// Mitsubishi GX Works2 project: ex2automation   PLC: FX3G

// global labels: Global1
VAR_GLOBAL
  start_switch AT X007 : BOOL;
  workday_start AT Y000 : BOOL;
  kill_switch AT X005 : BOOL;
  oatmeal_overr AT M0 : BOOL;
  protein_over AT M1 : BOOL;
  honey_over AT M2 : BOOL;
  dayover AT M3 : BOOL;
  daylight AT Y000 : BOOL;
  input_quantities AT X003 : BOOL;
  typeOfSnack AT X003 : BOOL;
END_VAR
VAR_GLOBAL CONSTANT
  const1 : INT := 2000;
END_VAR
VAR_GLOBAL
  normal_Snack AT M4 : BOOL;
  reset : BOOL;
  reset_Button AT M69 : BOOL;
  hold_Normal AT M41 : BOOL;
END_VAR
VAR_GLOBAL CONSTANT
  const2 : INT := 4000;
END_VAR
VAR_GLOBAL
  protein_Snack AT M5 : BOOL;
  hold_Protein AT M51 : BOOL;
  input_Oatmeal AT D1111 : REAL;
  oatmeal_Inv AT D1122 : REAL;
  input_protein AT D2222 : REAL;
  protein_Inv AT D2233 : REAL;
  input_Honey AT D3333 : REAL;
  honey_Inv AT D3344 : REAL;
  analog_input2 AT D8280 : INT;
END_VAR
VAR_GLOBAL CONSTANT
  const3 : REAL := 400;
  const4 : REAL := 320;
  const6 : REAL := 400;
  const7 : REAL := 320;
  const8 : REAL := 160;
  const9 : INT := 120;
END_VAR
VAR_GLOBAL
  start_shake_normal AT M10 : BOOL;
  start_shake_special AT M11 : BOOL;
  shakeTimer AT TC1 : BOOL;
END_VAR
VAR_GLOBAL CONSTANT
  shakeTimeValue : INT := 50;
END_VAR
VAR_GLOBAL
  timer_shake AT TS1 : BOOL;
  mixing_light AT Y003 : BOOL;
END_VAR
VAR_GLOBAL CONSTANT
  const5 : REAL := 160;
END_VAR
VAR_GLOBAL
  oatmeal_ok_n AT M42 : BOOL;
  protein_ok_n AT M43 : BOOL;
  honey_ok_n AT M44 : BOOL;
END_VAR
VAR_GLOBAL CONSTANT
  const0 : INT;
END_VAR
VAR_GLOBAL
  oatmeal_ok_p AT M52 : BOOL;
  protein_ok_p AT M53 : BOOL;
  honey_ok_p AT M54 : BOOL;
  func_reset AT M99 : BOOL;
  typeOfSnackHelp AT M33 : BOOL;
  hold_Shake AT M110 : BOOL;
  Bake_start AT X002 : BOOL;
  Bake_normal AT TC2 : BOOL;
  Bake_Protein AT TC3 : BOOL;
END_VAR
VAR_GLOBAL CONSTANT
  normalBakingTime : INT := 40;
  proteinBakingTime : INT := 50;
END_VAR
VAR_GLOBAL
  Baking_timer_normal AT TS2 : BOOL;
  Baking_timer_protein AT TS3 : BOOL;
  Bake_blink_help AT M60 : BOOL;
  blinkLight1 AT TC5 : BOOL;
END_VAR
VAR_GLOBAL CONSTANT
  blink_const : INT := 2;
END_VAR
VAR_GLOBAL
  blinktimer1 AT TS5 : BOOL;
  blinking_light1 AT Y001 : BOOL;
  blinkLight2 AT TC6 : BOOL;
  blinktime2 AT TS6 : BOOL;
  blinking_light2 AT Y002 : BOOL;
  packing_start AT X006 : BOOL;
  single_pack AT X000 : BOOL;
  light_help AT M61 : BOOL;
  packCounter AT CC1 : BOOL;
END_VAR
VAR_GLOBAL CONSTANT
  packconstant : INT := 8;
END_VAR
VAR_GLOBAL
  outPackCounter AT CS1 : BOOL;
  packinglight AT Y004 : BOOL;
END_VAR
VAR_GLOBAL CONSTANT
  const11 : INT := 1;
END_VAR
VAR_GLOBAL
  finishPackage AT D4444 : INT;
END_VAR
VAR_GLOBAL CONSTANT
  const12 : INT := 40;
END_VAR
VAR_GLOBAL
  analog_output AT D8282 : INT;
  reset_help AT M70 : BOOL;
  hold_bake_start AT M22 : BOOL;
END_VAR

// task Task_01 (event TRUE, interval 0, priority 31): POU_01

PROGRAM POU_01
(* structured ladder/FBD written out as ST: instructions are called as NAME(EN, inputs, outputs); _pN, _eN, _tN stand for wires *)
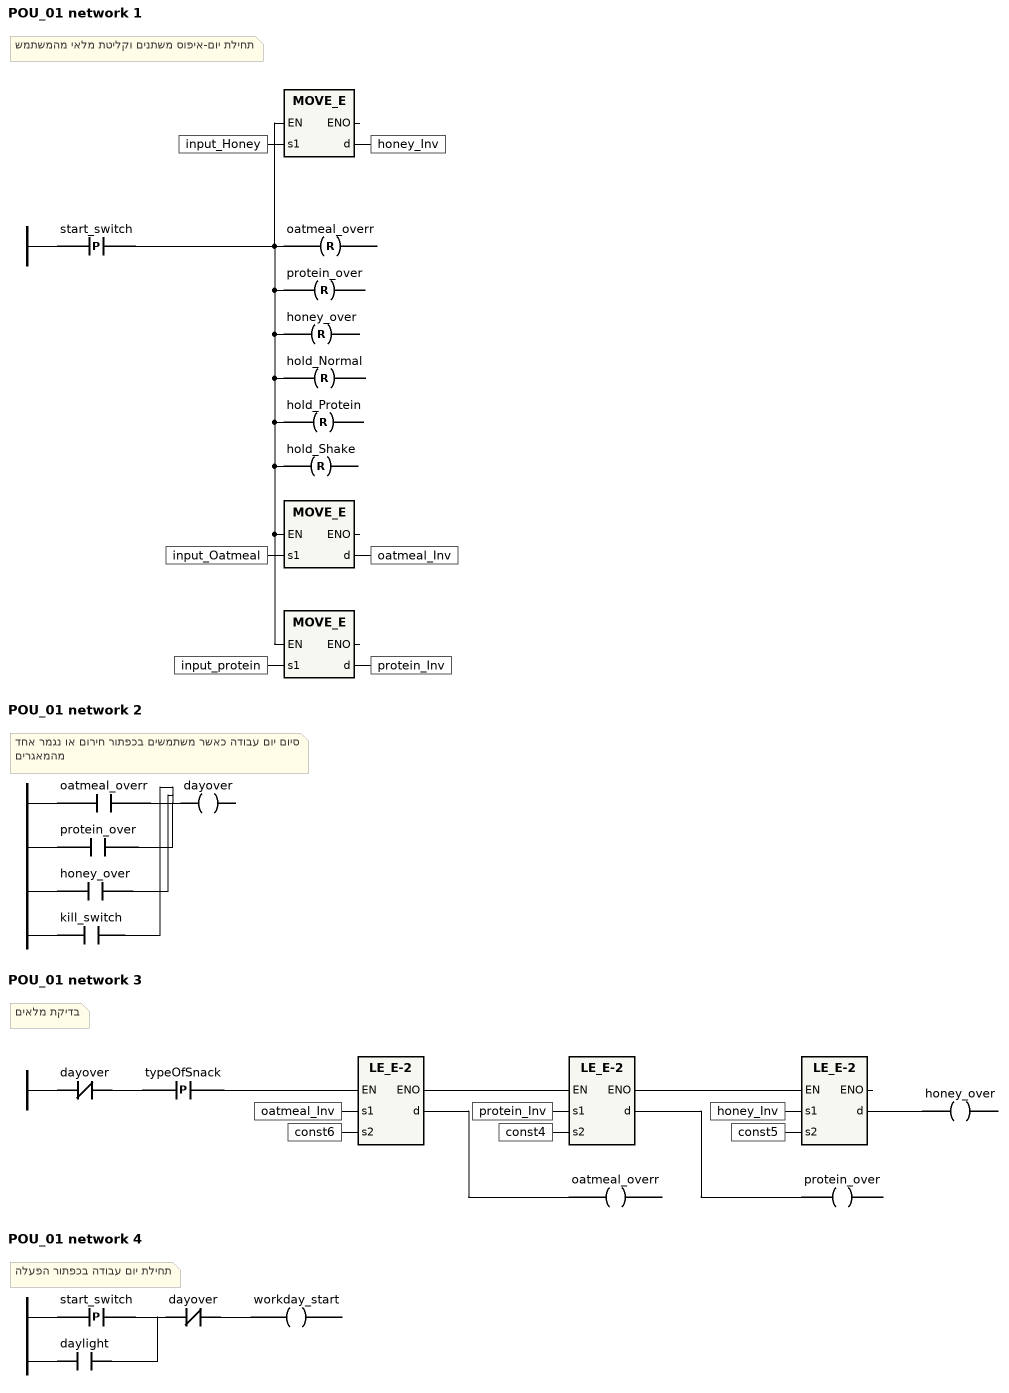
(* network 1 *)
(* תחילת יום-איפוס משתנים וקליטת מלאי מהמשתמש *)
_p1 := LDP(TRUE, start_switch);
RST(_p1, oatmeal_overr);
RST(_p1, protein_over);
MOVE_E(_p1, input_Honey, honey_Inv);
RST(_p1, honey_over);
RST(_p1, hold_Normal);
RST(_p1, hold_Protein);
RST(_p1, hold_Shake);
MOVE_E(_p1, input_Oatmeal, oatmeal_Inv);
MOVE_E(_p1, input_protein, protein_Inv);
(* network 2 *)
(* סיום יום עבודה כאשר משתמשים בכפתור חירום או נגמר אחד מהמאגרים *)
dayover := oatmeal_overr OR protein_over OR honey_over OR kill_switch;
(* network 3 *)
(* בדיקת מלאים *)
_e2 := LE_E(NOT dayover AND LDP(TRUE, typeOfSnack), oatmeal_Inv, const6, _t1);
_e4 := LE_E(_e2, protein_Inv, const4, _t3);
LE_E(_e4, honey_Inv, const5, _t5);
honey_over := _t5;
oatmeal_overr := _t1;
protein_over := _t3;
(* network 4 *)
(* תחילת יום עבודה בכפתור הפעלה *)
workday_start := (LDP(TRUE, start_switch) OR daylight) AND NOT dayover;
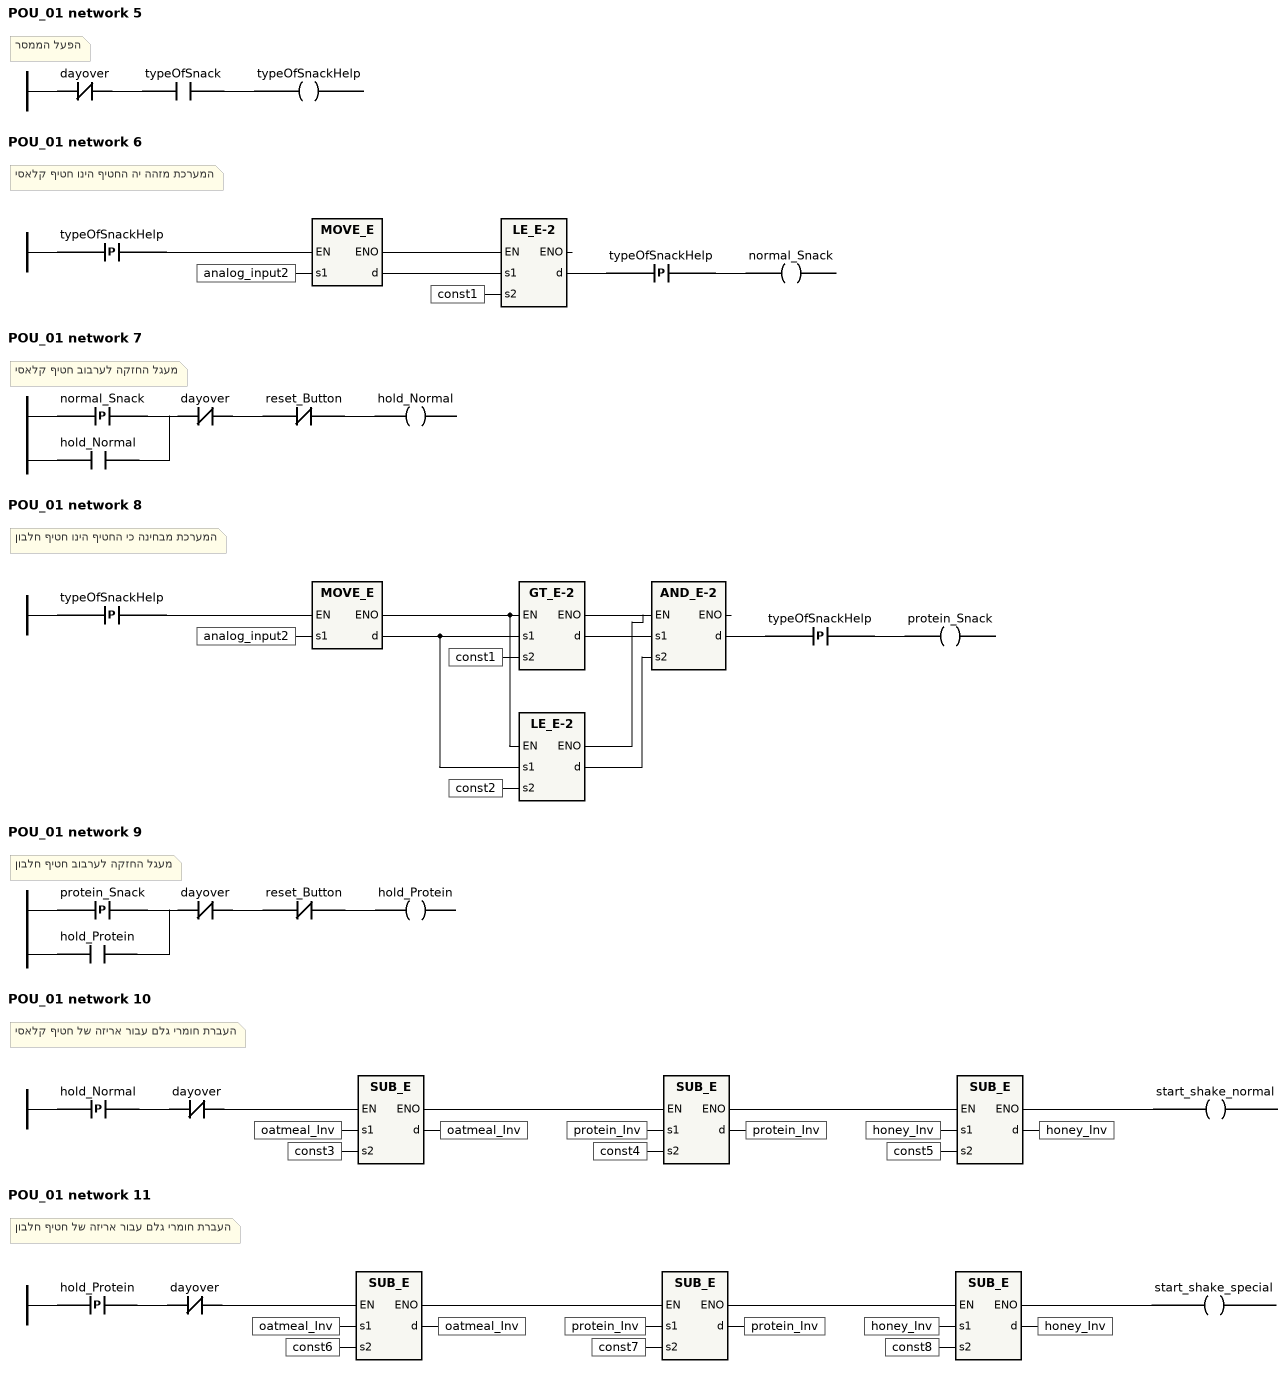
(* network 5 *)
(* הפעל הממסר *)
typeOfSnackHelp := NOT dayover AND typeOfSnack;
(* network 6 *)
(* המערכת מזהה יה החטיף הינו חטיף קלאסי *)
_e2 := MOVE_E(LDP(TRUE, typeOfSnackHelp), analog_input2, _t1);
LE_E(_e2, _t1, const1, _t3);
normal_Snack := _t3 AND LDP(TRUE, typeOfSnackHelp);
(* network 7 *)
(* מעגל החזקה לערבוב חטיף קלאסי *)
hold_Normal := ((LDP(TRUE, normal_Snack) OR hold_Normal) AND NOT dayover) AND NOT reset_Button;
(* network 8 *)
(* המערכת מבחינה כי החטיף הינו חטיף חלבון *)
_e2 := MOVE_E(LDP(TRUE, typeOfSnackHelp), analog_input2, _t1);
_e4 := GT_E(_e2, _t1, const1, _t3);
_e6 := LE_E(_e2, _t1, const2, _t5);
AND_E(_e4 OR _e6, _t3, _t5, _t7);
protein_Snack := _t7 AND LDP(TRUE, typeOfSnackHelp);
(* network 9 *)
(* מעגל החזקה לערבוב חטיף חלבון *)
hold_Protein := ((LDP(TRUE, protein_Snack) OR hold_Protein) AND NOT dayover) AND NOT reset_Button;
(* network 10 *)
(* העברת חומרי גלם עבור אריזה של חטיף קלאסי *)
_e1 := SUB_E(LDP(TRUE, hold_Normal) AND NOT dayover, oatmeal_Inv, const3, oatmeal_Inv);
_e2 := SUB_E(_e1, protein_Inv, const4, protein_Inv);
_e3 := SUB_E(_e2, honey_Inv, const5, honey_Inv);
start_shake_normal := _e3;
(* network 11 *)
(* העברת חומרי גלם עבור אריזה של חטיף חלבון *)
_e1 := SUB_E(LDP(TRUE, hold_Protein) AND NOT dayover, oatmeal_Inv, const6, oatmeal_Inv);
_e2 := SUB_E(_e1, protein_Inv, const7, protein_Inv);
_e3 := SUB_E(_e2, honey_Inv, const8, honey_Inv);
start_shake_special := _e3;
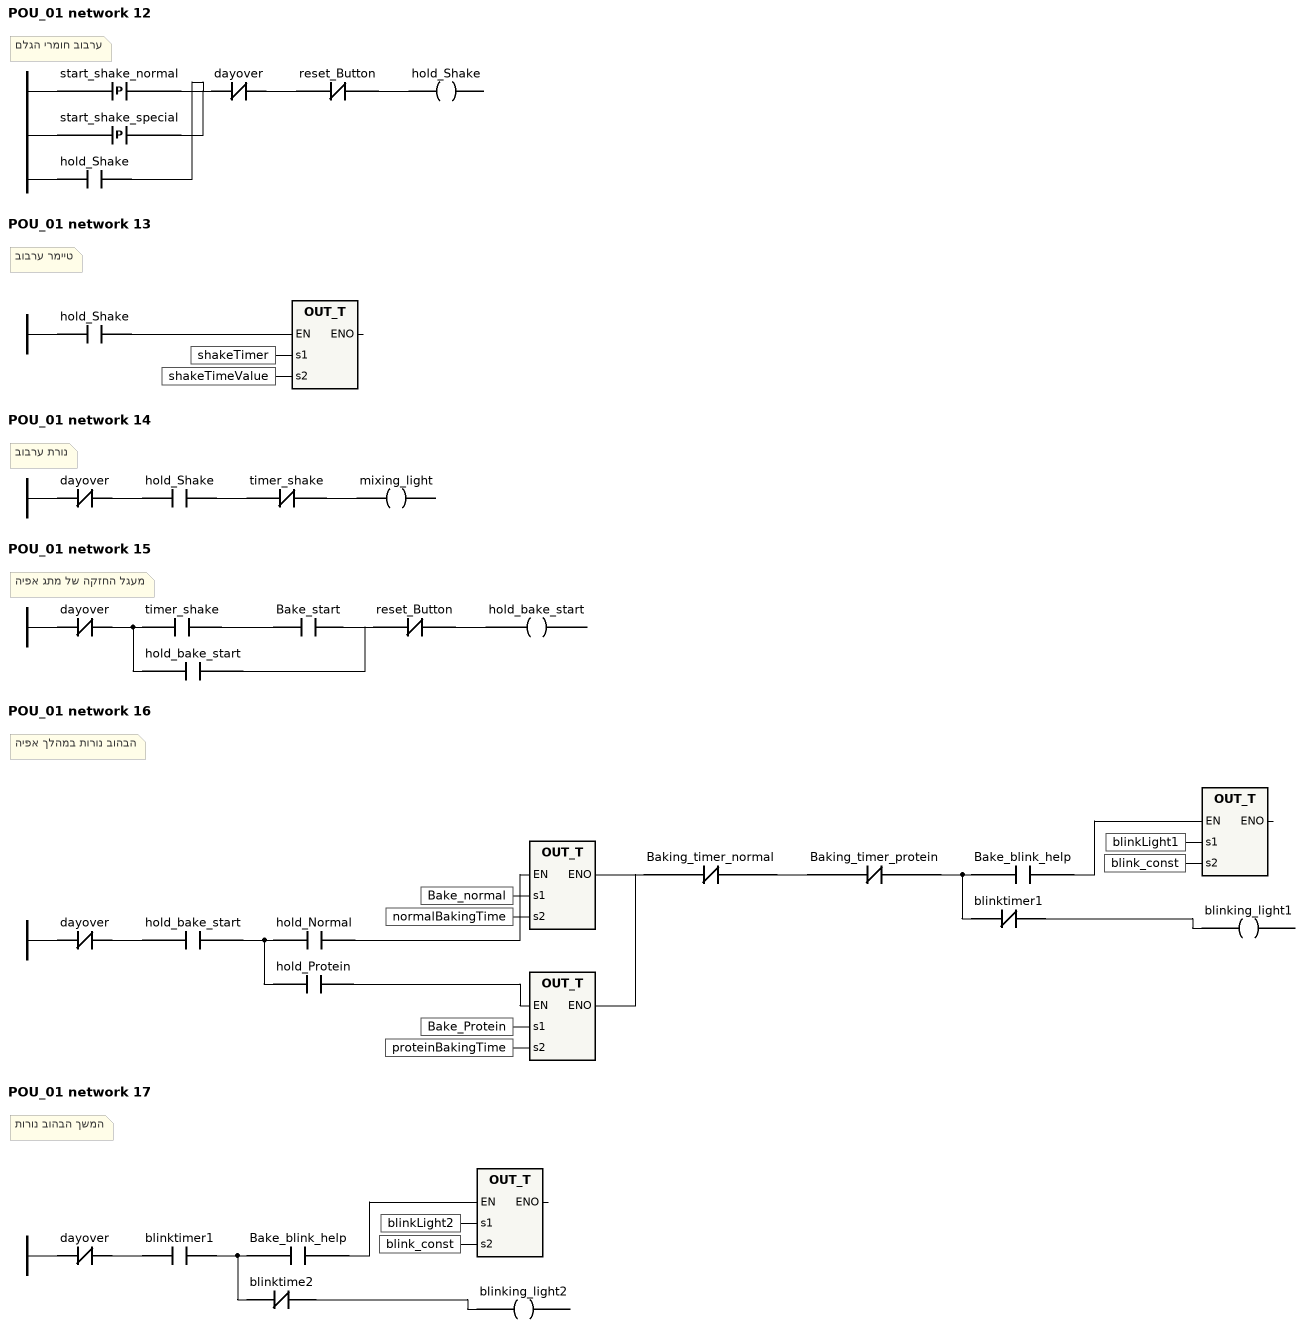
(* network 12 *)
(* ערבוב חומרי הגלם *)
hold_Shake := ((LDP(TRUE, start_shake_normal) OR LDP(TRUE, start_shake_special) OR hold_Shake) AND NOT dayover) AND NOT reset_Button;
(* network 13 *)
(* טיימר ערבוב *)
OUT_T(hold_Shake, shakeTimer, shakeTimeValue);
(* network 14 *)
(* נורת ערבוב *)
mixing_light := NOT dayover AND hold_Shake AND NOT timer_shake;
(* network 15 *)
(* מעגל החזקה של מתג אפיה *)
_p1 := NOT dayover;
hold_bake_start := ((_p1 AND timer_shake AND Bake_start) OR (_p1 AND hold_bake_start)) AND NOT reset_Button;
(* network 16 *)
(* הבהוב נורות במהלך אפיה *)
_p1 := NOT dayover AND hold_bake_start;
_e2 := OUT_T(_p1 AND hold_Normal, Bake_normal, normalBakingTime);
_e3 := OUT_T(_p1 AND hold_Protein, Bake_Protein, proteinBakingTime);
_p4 := ((_e2 OR _e3) AND NOT Baking_timer_normal) AND NOT Baking_timer_protein;
OUT_T(_p4 AND Bake_blink_help, blinkLight1, blink_const);
blinking_light1 := _p4 AND NOT blinktimer1;
(* network 17 *)
(* המשך הבהוב נורות *)
_p1 := NOT dayover AND blinktimer1;
OUT_T(_p1 AND Bake_blink_help, blinkLight2, blink_const);
blinking_light2 := _p1 AND NOT blinktime2;
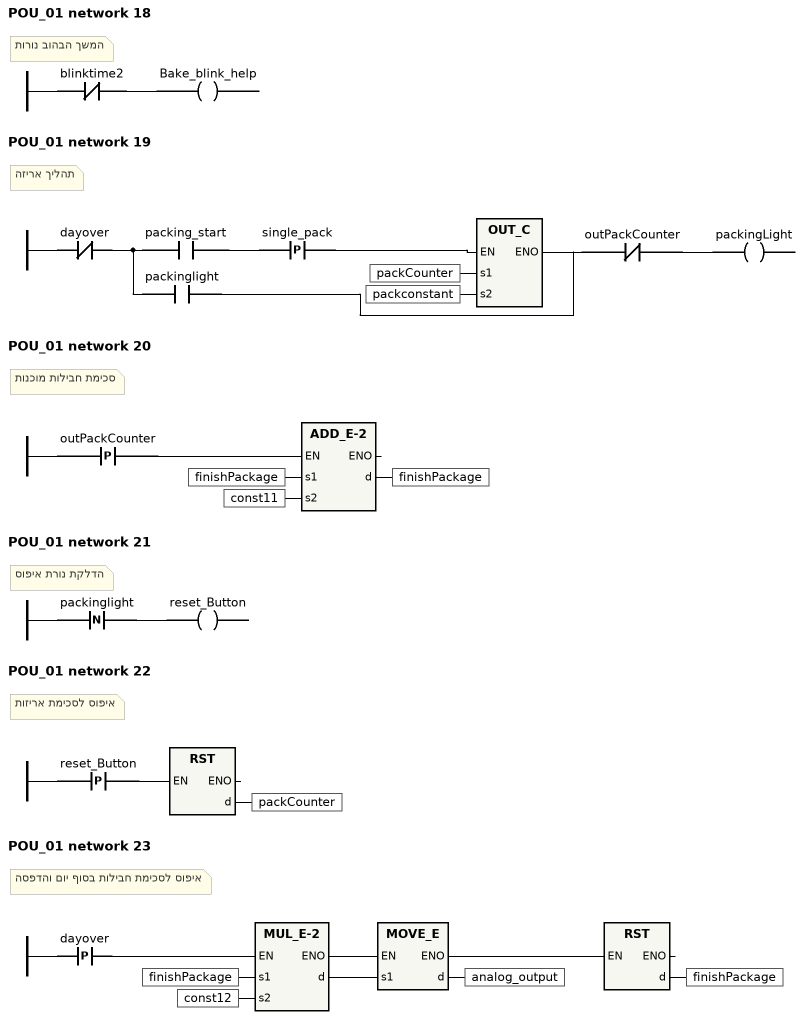
(* network 18 *)
(* המשך הבהוב נורות *)
Bake_blink_help := NOT blinktime2;
(* network 19 *)
(* תהליך אריזה *)
_p1 := NOT dayover;
_e2 := OUT_C(_p1 AND packing_start AND LDP(TRUE, single_pack), packCounter, packconstant);
packingLight := (_e2 OR (_p1 AND packinglight)) AND NOT outPackCounter;
(* network 20 *)
(* סכימת חבילות מוכנות *)
ADD_E(LDP(TRUE, outPackCounter), finishPackage, const11, finishPackage);
(* network 21 *)
(* הדלקת נורת איפוס *)
reset_Button := LDF(TRUE, packinglight);
(* network 22 *)
(* איפוס לסכימת אריזות *)
RST(LDP(TRUE, reset_Button), packCounter);
(* network 23 *)
(* איפוס לסכימת חבילות בסוף יום והדפסה *)
_e2 := MUL_E(LDP(TRUE, dayover), finishPackage, const12, _t1);
_e3 := MOVE_E(_e2, _t1, analog_output);
RST(_e3, finishPackage);
END_PROGRAM
